(* IEC 61131-3 sources: simple-control-modules/src/Encoder, 6 files *)

(* ---- CountMode.st ---- *)
NAMESPACE Simatic.Ax.SimpleControlModules
    TYPE
        CountMode : (Forward, Reverse) := Forward;
    END_TYPE
END_NAMESPACE

(* ---- Direction.st ---- *)
NAMESPACE Simatic.Ax.SimpleControlModules
    TYPE
        Direction : (Forward, Reverse, Undefined) := Forward;
    END_TYPE
END_NAMESPACE

(* ---- IEncoder.st ---- *)
NAMESPACE Simatic.Ax.SimpleControlModules
    INTERFACE IEncoder
        METHOD Evaluate
        END_METHOD
        METHOD Reset
        END_METHOD
        METHOD SetValue
            VAR_INPUT
                value : DINT;
            END_VAR
        END_METHOD
        METHOD GetValue : DINT
        END_METHOD
        METHOD SetDirection
            VAR_INPUT
                mode : CountMode;
            END_VAR
        END_METHOD
        METHOD RelativeCount : DINT
        END_METHOD
        METHOD ResetRelative
        END_METHOD
        METHOD GetModulo : DINT
        END_METHOD
    END_INTERFACE
END_NAMESPACE

(* ---- AbstractEncoder.st ---- *)
USING Simatic.Ax.Io.Input;
NAMESPACE Simatic.Ax.SimpleControlModules
    /// <summary>
    /// Class to handle a counter with an A and B signal
    /// </summary>
    CLASS ABSTRACT AbstractEncoder IMPLEMENTS IEncoder

        VAR PUBLIC
            Modulo : LINT := LINT#9223372036854775807;
        END_VAR

        VAR PROTECTED
            _encoderHasMoved : BOOL;
            _countMode : CountMode;
            _actualDirection : Direction;
            _encoderAbsCounter : Counter;
            _encoderRelativeCounter : Counter;
        END_VAR

        /// Reset encoder position to zero
        METHOD PUBLIC Reset
            _encoderAbsCounter.SetCounterValue(LINT#0);
            _encoderRelativeCounter.SetCounterValue(LINT#0);
            _actualDirection := Direction#Undefined;
        END_METHOD

        /// Set encoder to specific position
        /// value : Position which is set
        METHOD PUBLIC SetValue
            VAR_INPUT
                value : LINT;
            END_VAR
                _encoderAbsCounter.SetCounterValue(value := value);
                _encoderRelativeCounter.SetCounterValue(value := 0);
        END_METHOD

        /// Returns the actual encoder position
        /// Actual encoder position
        METHOD PUBLIC GetValue : LINT
            GetValue := _encoderAbsCounter.CounterValue() MOD Modulo;
        END_METHOD

        /// Evaluate encoder signals
        METHOD PUBLIC ABSTRACT Evaluate
        END_METHOD

        /// Returns if the encoder has moved
        /// Encoder has moved
        METHOD PUBLIC HasMoved : BOOL
            HasMoved := _encoderHasMoved;
            _encoderHasMoved := FALSE;
        END_METHOD

        /// Counts the relative pulses since the last Reset or ResetRelative command
        METHOD PUBLIC RelativeCount : LINT
            RelativeCount := _encoderRelativeCounter.CounterValue() MOD Modulo;
        END_METHOD

        /// Reset the relative counter
        METHOD PUBLIC ResetRelative
            _encoderRelativeCounter.SetCounterValue(LINT#0);
        END_METHOD

        METHOD PUBLIC SetDirection
            VAR_INPUT
                mode : CountMode;
            END_VAR
            _countMode := mode;
        END_METHOD

        METHOD PUBLIC GetModulo : LINT
            GetModulo := Modulo;
        END_METHOD
END_CLASS
END_NAMESPACE

(* ---- EncoderA.st ---- *)
USING Simatic.Ax.IO.Input;

NAMESPACE Simatic.Ax.SimpleControlModules

    /// Class to handle a counter with an A signal
    CLASS EncoderA EXTENDS AbstractEncoder

        VAR PUBLIC
            SignalA : ItfBinSignal;
        END_VAR

        /// Evaluate encoder signal A
        METHOD PUBLIC OVERRIDE Evaluate

            IF (THIS.ForwardPulse(SignalA)) THEN
                IF (_countMode = CountMode#FORWARD) THEN
                    _encoderAbsCounter.CountForward();
                    _encoderRelativeCounter.CountForward();
                ELSE
                    _encoderAbsCounter.CountReverse();
                    _encoderRelativeCounter.CountReverse();
                END_IF;
            END_IF;

        END_METHOD

        /// Returns if the encoder made a pulse
        /// A : A signal from encoder
        METHOD ForwardPulse : BOOL
            VAR_INPUT
                A : ItfBinSignal;
            END_VAR
            ForwardPulse := A.QRis() OR A.QFal();
        END_METHOD

    END_CLASS
END_NAMESPACE

(* ---- EncoderAB.st ---- *)
USING Simatic.Ax.IO.Input;
NAMESPACE Simatic.Ax.SimpleControlModules
    /// <summary>
    /// Class to handle a counter with an A and B signal
    /// </summary>
    CLASS EncoderAB EXTENDS AbstractEncoder
        VAR PUBLIC
            SignalA : ItfBinSignal;
            SignalB : ItfBinSignal;
        END_VAR

        /// Evaluate encoder for A B track
        METHOD PUBLIC OVERRIDE Evaluate

            VAR_TEMP
                _A : ItfBinSignal;
                _B : ItfBinSignal;
            END_VAR
            IF (_countMode = CountMode#Forward) THEN
                _A := SignalA;
                _B := SignalB;
            ELSE
                _A := SignalB;
                _B := SignalA;
            END_IF;

            IF (THIS.ForwardPulse(_A, _B)) THEN
                _encoderHasMoved := TRUE;
                _actualDirection := Direction#FORWARD;
                _encoderAbsCounter.CountForward();
                _encoderRelativeCounter.CountForward();
            //Reverse detection
            ELSIF (THIS.ReversePulse(_A, _B)) THEN
                _encoderHasMoved := TRUE;
                _actualDirection := Direction#REVERSE;
                _encoderAbsCounter.CountReverse();
                _encoderRelativeCounter.CountReverse();
            ELSE
                _actualDirection := Direction#FORWARD;
            END_IF;

        END_METHOD

        /// Pulse for two direction evaluation
        /// A : A signal from encoder
        /// B : B signal from encoder
        /// Returns Encoder signal A and/or B made pulse forward
        METHOD ForwardPulse : BOOL
            VAR_INPUT
                A : ItfBinSignal;
                B : ItfBinSignal;
            END_VAR
            ForwardPulse := A.QRis() AND NOT(B.Q())
                OR A.Q() AND B.QRis()
                OR A.QFal() AND B.Q()
                OR NOT(A.Q()) AND B.qFal();
        END_METHOD

        /// Pulse for two direction evaluation
        /// A : A signal from encoder
        /// B : B signal from encoder
        /// Returns Encoder signal A and/or B made pulse reverse
        METHOD ReversePulse : BOOL
            VAR_INPUT
                A : ItfBinSignal;
                B : ItfBinSignal;
            END_VAR
            ReversePulse := A.QRis() AND B.Q()
                OR NOT(A.Q()) AND B.QRis()
                OR A.QFal() AND NOT(B.Q())
                OR A.Q() AND B.qFal();
        END_METHOD

    END_CLASS
END_NAMESPACE
